    |   movel([0.490006, -1.325521, -2.603775, -0.783093, 1.570796, 2.060802],accel_mss,speed_ms,0,blend_radius_m)
    |   movel([0.490561, -1.327919, -2.602258, -0.782211, 1.570796, 2.061357],accel_mss,speed_ms,0,blend_radius_m)
    |   movel([0.493292, -1.324819, -2.604218, -0.783352, 1.570796, 2.064088],accel_mss,speed_ms,0,blend_radius_m)
    |   movel([0.496193, -1.321984, -2.605999, -0.784406, 1.570796, 2.066989],accel_mss,speed_ms,0,blend_radius_m)
    |   movel([0.499235, -1.319428, -2.607595, -0.785366, 1.570796, 2.070031],accel_mss,speed_ms,0,blend_radius_m)
    |   movel([0.502386, -1.317162, -2.609003, -0.786224, 1.570796, 2.073182],accel_mss,speed_ms,0,blend_radius_m)
    |   movel([0.505611, -1.315198, -2.610217, -0.786973, 1.570796, 2.076407],accel_mss,speed_ms,0,blend_radius_m)
    |   movel([0.508883, -1.313549, -2.611234, -0.787606, 1.570796, 2.079679],accel_mss,speed_ms,0,blend_radius_m)
    |   movel([0.512165, -1.312228, -2.612045, -0.788116, 1.570796, 2.082962],accel_mss,speed_ms,0,blend_radius_m)
    |   movel([0.515427, -1.311244, -2.612648, -0.788497, 1.570796, 2.086224],accel_mss,speed_ms,0,blend_radius_m)
    |   movel([0.518637, -1.310607, -2.613038, -0.788745, 1.570796, 2.089433],accel_mss,speed_ms,0,blend_radius_m)
    |   movel([0.521755, -1.310327, -2.613208, -0.788853, 1.570796, 2.092552],accel_mss,speed_ms,0,blend_radius_m)
    |   movel([0.524757, -1.310411, -2.613157, -0.788821, 1.570796, 2.095554],accel_mss,speed_ms,0,blend_radius_m)
    |   movel([0.527609, -1.310865, -2.612880, -0.788644, 1.570796, 2.098405],accel_mss,speed_ms,0,blend_radius_m)
    |   movel([0.530273, -1.311699, -2.612369, -0.788321, 1.570796, 2.101069],accel_mss,speed_ms,0,blend_radius_m)
    |   movel([0.532724, -1.312918, -2.611621, -0.787850, 1.570796, 2.103520],accel_mss,speed_ms,0,blend_radius_m)
    |   movel([0.534931, -1.314523, -2.610634, -0.787232, 1.570796, 2.105727],accel_mss,speed_ms,0,blend_radius_m)
    |   movel([0.536862, -1.316516, -2.609403, -0.786470, 1.570796, 2.107659],accel_mss,speed_ms,0,blend_radius_m)
    |   movel([0.538179, -1.318406, -2.608230, -0.785752, 1.570796, 2.108975],accel_mss,speed_ms,0,blend_radius_m)
    |   movel([0.539188, -1.320426, -2.606973, -0.784990, 1.570796, 2.109985],accel_mss,speed_ms,0,blend_radius_m)
    |   movel([0.539900, -1.322560, -2.605637, -0.784191, 1.570796, 2.110697],accel_mss,speed_ms,0,blend_radius_m)
    |   movel([0.540333, -1.324790, -2.604236, -0.783363, 1.570796, 2.111129],accel_mss,speed_ms,0,blend_radius_m)
    |   movel([0.540418, -1.329463, -2.601277, -0.781648, 1.570796, 2.111215],accel_mss,speed_ms,0,blend_radius_m)
    |   movel([0.539552, -1.334306, -2.598181, -0.779902, 1.570796, 2.110349],accel_mss,speed_ms,0,blend_radius_m)
    |   movel([0.537852, -1.339189, -2.595026, -0.778174, 1.570796, 2.108648],accel_mss,speed_ms,0,blend_radius_m)
    |   movel([0.535425, -1.343980, -2.591899, -0.776510, 1.570796, 2.106221],accel_mss,speed_ms,0,blend_radius_m)
    |   movel([0.532371, -1.348563, -2.588878, -0.774947, 1.570796, 2.103168],accel_mss,speed_ms,0,blend_radius_m)
    |   movel([0.528798, -1.352820, -2.586047, -0.773522, 1.570796, 2.099595],accel_mss,speed_ms,0,blend_radius_m)
    |   movel([0.524795, -1.356639, -2.583485, -0.772265, 1.570796, 2.095591],accel_mss,speed_ms,0,blend_radius_m)
    |   movel([0.520453, -1.359910, -2.581275, -0.771204, 1.570796, 2.091250],accel_mss,speed_ms,0,blend_radius_m)
    |   movel([0.515861, -1.362529, -2.579494, -0.770365, 1.570796, 2.086657],accel_mss,speed_ms,0,blend_radius_m)
    |   movel([0.513494, -1.363560, -2.578791, -0.770038, 1.570796, 2.084290],accel_mss,speed_ms,0,blend_radius_m)
    |   movel([0.511095, -1.364389, -2.578224, -0.769776, 1.570796, 2.081891],accel_mss,speed_ms,0,blend_radius_m)
    |   movel([0.508673, -1.364997, -2.577808, -0.769584, 1.570796, 2.079469],accel_mss,speed_ms,0,blend_radius_m)
    |   movel([0.506236, -1.365377, -2.577547, -0.769464, 1.570796, 2.077032],accel_mss,speed_ms,0,blend_radius_m)
    |   movel([0.503793, -1.365512, -2.577455, -0.769422, 1.570796, 2.074590],accel_mss,speed_ms,0,blend_radius_m)
    |   movel([0.501355, -1.365389, -2.577539, -0.769461, 1.570796, 2.072151],accel_mss,speed_ms,0,blend_radius_m)
    |   movel([0.498931, -1.364990, -2.577813, -0.769586, 1.570796, 2.069727],accel_mss,speed_ms,0,blend_radius_m)
    |   movel([0.496529, -1.364305, -2.578282, -0.769802, 1.570796, 2.067325],accel_mss,speed_ms,0,blend_radius_m)
    |   movel([0.494155, -1.363317, -2.578957, -0.770115, 1.570796, 2.064951],accel_mss,speed_ms,0,blend_radius_m)
    |   movel([0.491822, -1.362010, -2.579848, -0.770531, 1.570796, 2.062619],accel_mss,speed_ms,0,blend_radius_m)
    |   movel([0.490227, -1.360613, -2.580798, -0.770978, 1.570796, 2.061023],accel_mss,speed_ms,0,blend_radius_m)
    |   movel([0.486318, -1.356256, -2.583743, -0.772390, 1.570796, 2.057115],accel_mss,speed_ms,0,blend_radius_m)
    |   movel([0.483901, -1.352883, -2.586004, -0.773501, 1.570796, 2.054697],accel_mss,speed_ms,0,blend_radius_m)
    |   movel([0.481393, -1.348660, -2.588814, -0.774915, 1.570796, 2.052189],accel_mss,speed_ms,0,blend_radius_m)
    |   movel([0.478957, -1.343540, -2.592188, -0.776662, 1.570796, 2.049753],accel_mss,speed_ms,0,blend_radius_m)
    |   movel([0.476768, -1.337466, -2.596143, -0.778780, 1.570796, 2.047564],accel_mss,speed_ms,0,blend_radius_m)
    |   movel([0.475658, -1.332933, -2.599062, -0.780394, 1.570796, 2.046454],accel_mss,speed_ms,0,blend_radius_m)
    |   movel([0.475114, -1.328563, -2.601850, -0.781976, 1.570796, 2.045910],accel_mss,speed_ms,0,blend_radius_m)
    |   movel([0.475073, -1.324370, -2.604501, -0.783518, 1.570796, 2.045869],accel_mss,speed_ms,0,blend_radius_m)
    |   movel([0.475474, -1.320373, -2.607006, -0.785010, 1.570796, 2.046270],accel_mss,speed_ms,0,blend_radius_m)
    |   movel([0.476255, -1.316582, -2.609362, -0.786445, 1.570796, 2.047051],accel_mss,speed_ms,0,blend_radius_m)
    |   movel([0.477343, -1.313021, -2.611558, -0.787810, 1.570796, 2.048139],accel_mss,speed_ms,0,blend_radius_m)
    |   movel([0.478674, -1.309707, -2.613587, -0.789095, 1.570796, 2.049470],accel_mss,speed_ms,0,blend_radius_m)
    |   movel([0.480175, -1.306660, -2.615440, -0.790289, 1.570796, 2.050971],accel_mss,speed_ms,0,blend_radius_m)
    |   movel([0.483403, -1.301447, -2.618581, -0.792361, 1.570796, 2.054199],accel_mss,speed_ms,0,blend_radius_m)
    |   movel([0.486444, -1.297538, -2.620914, -0.793937, 1.570796, 2.057241],accel_mss,speed_ms,0,blend_radius_m)
    |   movel([0.488705, -1.295089, -2.622365, -0.794935, 1.570796, 2.059502],accel_mss,speed_ms,0,blend_radius_m)
    |   movel([0.489590, -1.294242, -2.622865, -0.795281, 1.570796, 2.060387],accel_mss,speed_ms,0,blend_radius_m)
    |   movel([0.493944, -1.290499, -2.625065, -0.796825, 1.570796, 2.064741],accel_mss,speed_ms,0,blend_radius_m)
    |   movel([0.498273, -1.287334, -2.626911, -0.798144, 1.570796, 2.069069],accel_mss,speed_ms,0,blend_radius_m)
    |   movel([0.502541, -1.284718, -2.628427, -0.799244, 1.570796, 2.073337],accel_mss,speed_ms,0,blend_radius_m)
    |   movel([0.506719, -1.282608, -2.629643, -0.800137, 1.570796, 2.077516],accel_mss,speed_ms,0,blend_radius_m)
    |   movel([0.510774, -1.280967, -2.630586, -0.800836, 1.570796, 2.081570],accel_mss,speed_ms,0,blend_radius_m)
    |   movel([0.514673, -1.279752, -2.631281, -0.801356, 1.570796, 2.085470],accel_mss,speed_ms,0,blend_radius_m)
    |   movel([0.518397, -1.278914, -2.631760, -0.801715, 1.570796, 2.089193],accel_mss,speed_ms,0,blend_radius_m)
    |   movel([0.521908, -1.278413, -2.632046, -0.801930, 1.570796, 2.092705],accel_mss,speed_ms,0,blend_radius_m)
    |   movel([0.528205, -1.278218, -2.632156, -0.802014, 1.570796, 2.099001],accel_mss,speed_ms,0,blend_radius_m)
    |   movel([0.533373, -1.278773, -2.631841, -0.801776, 1.570796, 2.104170],accel_mss,speed_ms,0,blend_radius_m)
    |   movel([0.537237, -1.279670, -2.631328, -0.801391, 1.570796, 2.108033],accel_mss,speed_ms,0,blend_radius_m)
    |   movel([0.539631, -1.280510, -2.630848, -0.801031, 1.570796, 2.110427],accel_mss,speed_ms,0,blend_radius_m)
    |   movel([0.545351, -1.282444, -2.629738, -0.800207, 1.570796, 2.116147],accel_mss,speed_ms,0,blend_radius_m)
    |   movel([0.551208, -1.285055, -2.628232, -0.799102, 1.570796, 2.122004],accel_mss,speed_ms,0,blend_radius_m)
    |   movel([0.557042, -1.287887, -2.626589, -0.797913, 1.570796, 2.127839],accel_mss,speed_ms,0,blend_radius_m)
    |   movel([0.562712, -1.290482, -2.625075, -0.796832, 1.570796, 2.133508],accel_mss,speed_ms,0,blend_radius_m)
    |   movel([0.568089, -1.292385, -2.623959, -0.796045, 1.570796, 2.138885],accel_mss,speed_ms,0,blend_radius_m)
    |   movel([0.570630, -1.292931, -2.623638, -0.795820, 1.570796, 2.141426],accel_mss,speed_ms,0,blend_radius_m)
    |   movel([0.573054, -1.293131, -2.623520, -0.795738, 1.570796, 2.143850],accel_mss,speed_ms,0,blend_radius_m)
    |   movel([0.575351, -1.292924, -2.623642, -0.795823, 1.570796, 2.146147],accel_mss,speed_ms,0,blend_radius_m)
    |   movel([0.577504, -1.292250, -2.624039, -0.796101, 1.570796, 2.148300],accel_mss,speed_ms,0,blend_radius_m)
    |   movel([0.579504, -1.291047, -2.624744, -0.796598, 1.570796, 2.150301],accel_mss,speed_ms,0,blend_radius_m)
    |   movel([0.581338, -1.289257, -2.625791, -0.797341, 1.570796, 2.152134],accel_mss,speed_ms,0,blend_radius_m)
    |   movel([0.582452, -1.287733, -2.626679, -0.797977, 1.570796, 2.153249],accel_mss,speed_ms,0,blend_radius_m)
    |   movel([0.583281, -1.286224, -2.627555, -0.798610, 1.570796, 2.154077],accel_mss,speed_ms,0,blend_radius_m)
    |   movel([0.584194, -1.283247, -2.629276, -0.799866, 1.570796, 2.154991],accel_mss,speed_ms,0,blend_radius_m)
    |   movel([0.584298, -1.280332, -2.630949, -0.801107, 1.570796, 2.155094],accel_mss,speed_ms,0,blend_radius_m)
    |   movel([0.583810, -1.277482, -2.632576, -0.802331, 1.570796, 2.154606],accel_mss,speed_ms,0,blend_radius_m)
    |   movel([0.581965, -1.272012, -2.635669, -0.804708, 1.570796, 2.152761],accel_mss,speed_ms,0,blend_radius_m)
    |   movel([0.581068, -1.269398, -2.637134, -0.805858, 1.570796, 2.151864],accel_mss,speed_ms,0,blend_radius_m)
    |   movel([0.580496, -1.266865, -2.638545, -0.806979, 1.570796, 2.151293],accel_mss,speed_ms,0,blend_radius_m)
    |   movel([0.580460, -1.262675, -2.640863, -0.808852, 1.570796, 2.151256],accel_mss,speed_ms,0,blend_radius_m)
    |   movel([0.581118, -1.257317, -2.643795, -0.811277, 1.570796, 2.151914],accel_mss,speed_ms,0,blend_radius_m)
    |   movel([0.582306, -1.251758, -2.646801, -0.813831, 1.570796, 2.153102],accel_mss,speed_ms,0,blend_radius_m)
    |   movel([0.583843, -1.247006, -2.649341, -0.816042, 1.570796, 2.154640],accel_mss,speed_ms,0,blend_radius_m)
    |   movel([0.585406, -1.244036, -2.650914, -0.817438, 1.570796, 2.156203],accel_mss,speed_ms,0,blend_radius_m)
    |   movel([0.587619, -1.240418, -2.652818, -0.819153, 1.570796, 2.158415],accel_mss,speed_ms,0,blend_radius_m)
    |   movel([0.589696, -1.236967, -2.654618, -0.820803, 1.570796, 2.160493],accel_mss,speed_ms,0,blend_radius_m)
    |   movel([0.590831, -1.234525, -2.655885, -0.821979, 1.570796, 2.161628],accel_mss,speed_ms,0,blend_radius_m)
    |   movel([0.590982, -1.232123, -2.657123, -0.823143, 1.570796, 2.161779],accel_mss,speed_ms,0,blend_radius_m)
    |   movel([0.590662, -1.229442, -2.658497, -0.824449, 1.570796, 2.161458],accel_mss,speed_ms,0,blend_radius_m)
    |   movel([0.590352, -1.226433, -2.660030, -0.825926, 1.570796, 2.161148],accel_mss,speed_ms,0,blend_radius_m)
    |   movel([0.590532, -1.223054, -2.661739, -0.827596, 1.570796, 2.161328],accel_mss,speed_ms,0,blend_radius_m)
    |   movel([0.591130, -1.220931, -2.662806, -0.828652, 1.570796, 2.161926],accel_mss,speed_ms,0,blend_radius_m)
    |   speed_ms = 0.003
    |   movel([0.591130, -1.213790, -2.659255, -0.839344, 1.570796, 2.161926],accel_mss,speed_ms,0,blend_radius_m)
    |   speed_ms = 0.05
    |   movel([0.591130, -1.186616, -2.644793, -0.880980, 1.570796, 2.161926],accel_mss,speed_ms,0,blend_radius_m)
    |   #M_RunCode9
    |   movel([0.476665, -1.280558, -2.594852, -0.836979, 1.570796, 2.047461],accel_mss,speed_ms,0,blend_radius_m)
    |   #M_RunCode3
    |   movel([0.476665, -1.306620, -2.608077, -0.797692, 1.570796, 2.047461],accel_mss,speed_ms,0,blend_radius_m)
    |   speed_ms = 0.003
    |   movel([0.476665, -1.313420, -2.611313, -0.787656, 1.570796, 2.047461],accel_mss,speed_ms,0,blend_radius_m)
    |   speed_ms = 0.02
    |   movel([0.470649, -1.312090, -2.612129, -0.788169, 1.570796, 2.041445],accel_mss,speed_ms,0,blend_radius_m)
    |   movel([0.464562, -1.311541, -2.612466, -0.788382, 1.570796, 2.035358],accel_mss,speed_ms,0,blend_radius_m)
    |   movel([0.458473, -1.311678, -2.612382, -0.788329, 1.570796, 2.029269],accel_mss,speed_ms,0,blend_radius_m)
    |   movel([0.452461, -1.312404, -2.611937, -0.788048, 1.570796, 2.023258],accel_mss,speed_ms,0,blend_radius_m)
    |   movel([0.446593, -1.313618, -2.611191, -0.787580, 1.570796, 2.017390],accel_mss,speed_ms,0,blend_radius_m)
    |   movel([0.440937, -1.315226, -2.610200, -0.786963, 1.570796, 2.011733],accel_mss,speed_ms,0,blend_radius_m)
    |   movel([0.435558, -1.317124, -2.609026, -0.786238, 1.570796, 2.006355],accel_mss,speed_ms,0,blend_radius_m)
    |   movel([0.430517, -1.319217, -2.607726, -0.785446, 1.570796, 2.001314],accel_mss,speed_ms,0,blend_radius_m)
    |   movel([0.425875, -1.321405, -2.606361, -0.784623, 1.570796, 1.996671],accel_mss,speed_ms,0,blend_radius_m)
    |   movel([0.421681, -1.323599, -2.604985, -0.783804, 1.570796, 1.992477],accel_mss,speed_ms,0,blend_radius_m)
    |   movel([0.414869, -1.327618, -2.602449, -0.782322, 1.570796, 1.985665],accel_mss,speed_ms,0,blend_radius_m)
    |   movel([0.410490, -1.330547, -2.600587, -0.781255, 1.570796, 1.981286],accel_mss,speed_ms,0,blend_radius_m)
    |   movel([0.408940, -1.331678, -2.599865, -0.780846, 1.570796, 1.979736],accel_mss,speed_ms,0,blend_radius_m)
    |   movel([0.406435, -1.333398, -2.598764, -0.780227, 1.570796, 1.977231],accel_mss,speed_ms,0,blend_radius_m)
    |   movel([0.400082, -1.338331, -2.595582, -0.778475, 1.570796, 1.970878],accel_mss,speed_ms,0,blend_radius_m)
    |   movel([0.396014, -1.341882, -2.593272, -0.777235, 1.570796, 1.966810],accel_mss,speed_ms,0,blend_radius_m)
    |   movel([0.391649, -1.346090, -2.590512, -0.775787, 1.570796, 1.962445],accel_mss,speed_ms,0,blend_radius_m)
    |   movel([0.387205, -1.350897, -2.587329, -0.774163, 1.570796, 1.958001],accel_mss,speed_ms,0,blend_radius_m)
    |   movel([0.382897, -1.356249, -2.583747, -0.772392, 1.570796, 1.953693],accel_mss,speed_ms,0,blend_radius_m)
    |   movel([0.378940, -1.362087, -2.579796, -0.770506, 1.570796, 1.949736],accel_mss,speed_ms,0,blend_radius_m)
    |   movel([0.375536, -1.368352, -2.575501, -0.768535, 1.570796, 1.946332],accel_mss,speed_ms,0,blend_radius_m)
    |   movel([0.374104, -1.371628, -2.573234, -0.767527, 1.570796, 1.944900],accel_mss,speed_ms,0,blend_radius_m)
    |   movel([0.372885, -1.374989, -2.570892, -0.766508, 1.570796, 1.943682],accel_mss,speed_ms,0,blend_radius_m)
    |   movel([0.371898, -1.378433, -2.568475, -0.765481, 1.570796, 1.942695],accel_mss,speed_ms,0,blend_radius_m)
    |   movel([0.371171, -1.381949, -2.565991, -0.764449, 1.570796, 1.941968],accel_mss,speed_ms,0,blend_radius_m)
    |   movel([0.370725, -1.385536, -2.563438, -0.763416, 1.570796, 1.941522],accel_mss,speed_ms,0,blend_radius_m)
    |   movel([0.370579, -1.389183, -2.560823, -0.762383, 1.570796, 1.941375],accel_mss,speed_ms,0,blend_radius_m)
    |   movel([0.370755, -1.392891, -2.558144, -0.761354, 1.570796, 1.941551],accel_mss,speed_ms,0,blend_radius_m)
    |   movel([0.371275, -1.396654, -2.555406, -0.760329, 1.570796, 1.942071],accel_mss,speed_ms,0,blend_radius_m)
    |   movel([0.372155, -1.400470, -2.552608, -0.759311, 1.570796, 1.942952],accel_mss,speed_ms,0,blend_radius_m)
    |   movel([0.373415, -1.404335, -2.549753, -0.758301, 1.570796, 1.944212],accel_mss,speed_ms,0,blend_radius_m)
    |   movel([0.375074, -1.408244, -2.546843, -0.757303, 1.570796, 1.945870],accel_mss,speed_ms,0,blend_radius_m)
    |   movel([0.377150, -1.412202, -2.543872, -0.756314, 1.570796, 1.947946],accel_mss,speed_ms,0,blend_radius_m)
    |   movel([0.377336, -1.412494, -2.543653, -0.756242, 1.570796, 1.948133],accel_mss,speed_ms,0,blend_radius_m)
    |   movel([0.380023, -1.415995, -2.541005, -0.755389, 1.570796, 1.950819],accel_mss,speed_ms,0,blend_radius_m)
    |   movel([0.382798, -1.419057, -2.538674, -0.754658, 1.570796, 1.953595],accel_mss,speed_ms,0,blend_radius_m)
    |   movel([0.385653, -1.421704, -2.536648, -0.754037, 1.570796, 1.956449],accel_mss,speed_ms,0,blend_radius_m)
    |   movel([0.388573, -1.423964, -2.534910, -0.753515, 1.570796, 1.959369],accel_mss,speed_ms,0,blend_radius_m)
    |   movel([0.391553, -1.425859, -2.533447, -0.753083, 1.570796, 1.962350],accel_mss,speed_ms,0,blend_radius_m)
    |   movel([0.394582, -1.427414, -2.532242, -0.752733, 1.570796, 1.965378],accel_mss,speed_ms,0,blend_radius_m)
    |   movel([0.397649, -1.428652, -2.531281, -0.752456, 1.570796, 1.968446],accel_mss,speed_ms,0,blend_radius_m)
    |   movel([0.400745, -1.429592, -2.530549, -0.752248, 1.570796, 1.971541],accel_mss,speed_ms,0,blend_radius_m)
    |   movel([0.403861, -1.430257, -2.530030, -0.752101, 1.570796, 1.974657],accel_mss,speed_ms,0,blend_radius_m)
    |   movel([0.406983, -1.430669, -2.529709, -0.752011, 1.570796, 1.977780],accel_mss,speed_ms,0,blend_radius_m)
    |   movel([0.410106, -1.430846, -2.529570, -0.751972, 1.570796, 1.980902],accel_mss,speed_ms,0,blend_radius_m)
    |   movel([0.413214, -1.430810, -2.529598, -0.751980, 1.570796, 1.984011],accel_mss,speed_ms,0,blend_radius_m)
    |   movel([0.419348, -1.430180, -2.530091, -0.752118, 1.570796, 1.990145],accel_mss,speed_ms,0,blend_radius_m)
    |   movel([0.425295, -1.428930, -2.531064, -0.752394, 1.570796, 1.996092],accel_mss,speed_ms,0,blend_radius_m)
    |   movel([0.430960, -1.427223, -2.532390, -0.752775, 1.570796, 2.001756],accel_mss,speed_ms,0,blend_radius_m)
    |   movel([0.436239, -1.425214, -2.533946, -0.753229, 1.570796, 2.007035],accel_mss,speed_ms,0,blend_radius_m)
    |   movel([0.441026, -1.423063, -2.535604, -0.753722, 1.570796, 2.011822],accel_mss,speed_ms,0,blend_radius_m)
    |   movel([0.445211, -1.420929, -2.537243, -0.754217, 1.570796, 2.016007],accel_mss,speed_ms,0,blend_radius_m)
    |   movel([0.451296, -1.417374, -2.539957, -0.755058, 1.570796, 2.022092],accel_mss,speed_ms,0,blend_radius_m)
    |   movel([0.453539, -1.415886, -2.541087, -0.755415, 1.570796, 2.024335],accel_mss,speed_ms,0,blend_radius_m)
    |   movel([0.454914, -1.415023, -2.541742, -0.755624, 1.570796, 2.025710],accel_mss,speed_ms,0,blend_radius_m)
    |   movel([0.458633, -1.412486, -2.543658, -0.756244, 1.570796, 2.029430],accel_mss,speed_ms,0,blend_radius_m)
    |   movel([0.464103, -1.408343, -2.546768, -0.757278, 1.570796, 2.034900],accel_mss,speed_ms,0,blend_radius_m)
    |   movel([0.470740, -1.402647, -2.551003, -0.758740, 1.570796, 2.041536],accel_mss,speed_ms,0,blend_radius_m)
    |   movel([0.474312, -1.399227, -2.553522, -0.759640, 1.570796, 2.045108],accel_mss,speed_ms,0,blend_radius_m)
    |   movel([0.477954, -1.395435, -2.556295, -0.760659, 1.570796, 2.048750],accel_mss,speed_ms,0,blend_radius_m)
    |   movel([0.481594, -1.391266, -2.559321, -0.761802, 1.570796, 2.052390],accel_mss,speed_ms,0,blend_radius_m)
    |   movel([0.485155, -1.386723, -2.562589, -0.763078, 1.570796, 2.055951],accel_mss,speed_ms,0,blend_radius_m)
    |   movel([0.488560, -1.381808, -2.566091, -0.764491, 1.570796, 2.059356],accel_mss,speed_ms,0,blend_radius_m)
    |   movel([0.491732, -1.376516, -2.569822, -0.766051, 1.570796, 2.062528],accel_mss,speed_ms,0,blend_radius_m)
    |   movel([0.494590, -1.370849, -2.573774, -0.767765, 1.570796, 2.065387],accel_mss,speed_ms,0,blend_radius_m)
    |   movel([0.497047, -1.364802, -2.577941, -0.769645, 1.570796, 2.067843],accel_mss,speed_ms,0,blend_radius_m)
    |   speed_ms = 0.003
    |   movel([0.497047, -1.358244, -2.574877, -0.779268, 1.570796, 2.067843],accel_mss,speed_ms,0,blend_radius_m)
    |   speed_ms = 0.05
    |   movel([0.497047, -1.333023, -2.562333, -0.817033, 1.570796, 2.067843],accel_mss,speed_ms,0,blend_radius_m)
    |   #M_RunCode9
    |   movel([0.471807, -1.327561, -2.565883, -0.818945, 1.570796, 2.042603],accel_mss,speed_ms,0,blend_radius_m)
    |   #M_RunCode3
    |   # logo 1
    |   movel([0.471807, -1.352876, -2.578497, -0.781015, 1.570796, 2.042603],accel_mss,speed_ms,0,blend_radius_m)
    |   speed_ms = 0.003
    |   movel([0.471807, -1.359461, -2.581579, -0.771349, 1.570796, 2.042603],accel_mss,speed_ms,0,blend_radius_m)
    |   speed_ms = 0.007
    |   movel([0.469753, -1.361986, -2.579865, -0.770539, 1.570796, 2.040549],accel_mss,speed_ms,0,blend_radius_m)
    |   movel([0.467378, -1.364236, -2.578329, -0.769824, 1.570796, 2.038174],accel_mss,speed_ms,0,blend_radius_m)
    |   movel([0.464761, -1.366165, -2.577007, -0.769217, 1.570796, 2.035557],accel_mss,speed_ms,0,blend_radius_m)
    |   movel([0.461981, -1.367726, -2.575933, -0.768730, 1.570796, 2.032778],accel_mss,speed_ms,0,blend_radius_m)
    |   movel([0.459114, -1.368870, -2.575144, -0.768375, 1.570796, 2.029910],accel_mss,speed_ms,0,blend_radius_m)
    |   movel([0.456235, -1.369551, -2.574673, -0.768165, 1.570796, 2.027032],accel_mss,speed_ms,0,blend_radius_m)
    |   movel([0.453420, -1.369720, -2.574557, -0.768113, 1.570796, 2.024216],accel_mss,speed_ms,0,blend_radius_m)
    |   movel([0.453380, -1.369716, -2.574559, -0.768114, 1.570796, 2.024176],accel_mss,speed_ms,0,blend_radius_m)
    |   movel([0.447352, -1.369503, -2.574707, -0.768180, 1.570796, 2.018149],accel_mss,speed_ms,0,blend_radius_m)
    |   movel([0.443007, -1.378673, -2.568306, -0.765410, 1.570796, 2.013804],accel_mss,speed_ms,0,blend_radius_m)
    |   movel([0.435809, -1.378470, -2.568449, -0.765470, 1.570796, 2.006605],accel_mss,speed_ms,0,blend_radius_m)
    |   movel([0.448034, -1.352401, -2.586327, -0.773661, 1.570796, 2.018830],accel_mss,speed_ms,0,blend_radius_m)
    |   movel([0.455424, -1.352614, -2.586184, -0.773591, 1.570796, 2.026221],accel_mss,speed_ms,0,blend_radius_m)
    |   movel([0.450911, -1.362037, -2.579830, -0.770522, 1.570796, 2.021708],accel_mss,speed_ms,0,blend_radius_m)
    |   movel([0.457056, -1.362252, -2.579683, -0.770454, 1.570796, 2.027852],accel_mss,speed_ms,0,blend_radius_m)
    |   movel([0.458332, -1.362171, -2.579738, -0.770479, 1.570796, 2.029128],accel_mss,speed_ms,0,blend_radius_m)
    |   movel([0.459648, -1.361851, -2.579957, -0.770582, 1.570796, 2.030444],accel_mss,speed_ms,0,blend_radius_m)
    |   movel([0.460964, -1.361314, -2.580321, -0.770753, 1.570796, 2.031760],accel_mss,speed_ms,0,blend_radius_m)
    |   movel([0.462242, -1.360591, -2.580813, -0.770985, 1.570796, 2.033038],accel_mss,speed_ms,0,blend_radius_m)
    |   movel([0.463445, -1.359699, -2.581418, -0.771272, 1.570796, 2.034241],accel_mss,speed_ms,0,blend_radius_m)
    |   movel([0.464532, -1.358666, -2.582117, -0.771606, 1.570796, 2.035329],accel_mss,speed_ms,0,blend_radius_m)
    |   movel([0.465466, -1.357515, -2.582895, -0.771979, 1.570796, 2.036262],accel_mss,speed_ms,0,blend_radius_m)
    |   movel([0.466207, -1.356275, -2.583730, -0.772384, 1.570796, 2.037003],accel_mss,speed_ms,0,blend_radius_m)
    |   movel([0.466698, -1.355017, -2.584575, -0.772796, 1.570796, 2.037494],accel_mss,speed_ms,0,blend_radius_m)
    |   movel([0.466925, -1.353822, -2.585377, -0.773190, 1.570796, 2.037721],accel_mss,speed_ms,0,blend_radius_m)
    |   movel([0.466616, -1.351745, -2.586764, -0.773880, 1.570796, 2.037412],accel_mss,speed_ms,0,blend_radius_m)
    |   movel([0.466103, -1.350922, -2.587312, -0.774155, 1.570796, 2.036899],accel_mss,speed_ms,0,blend_radius_m)
    |   movel([0.465361, -1.350281, -2.587739, -0.774369, 1.570796, 2.036158],accel_mss,speed_ms,0,blend_radius_m)
    |   movel([0.464402, -1.349855, -2.588022, -0.774512, 1.570796, 2.035199],accel_mss,speed_ms,0,blend_radius_m)
    |   movel([0.463240, -1.349675, -2.588141, -0.774573, 1.570796, 2.034037],accel_mss,speed_ms,0,blend_radius_m)
    |   movel([0.438898, -1.349022, -2.588575, -0.774793, 1.570796, 2.009694],accel_mss,speed_ms,0,blend_radius_m)
    |   movel([0.438801, -1.346776, -2.590060, -0.775553, 1.570796, 2.009597],accel_mss,speed_ms,0,blend_radius_m)
    |   movel([0.438301, -1.344731, -2.591406, -0.776252, 1.570796, 2.009097],accel_mss,speed_ms,0,blend_radius_m)
    |   movel([0.437406, -1.342923, -2.592592, -0.776875, 1.570796, 2.008203],accel_mss,speed_ms,0,blend_radius_m)
    |   movel([0.436133, -1.341382, -2.593598, -0.777408, 1.570796, 2.006929],accel_mss,speed_ms,0,blend_radius_m)
    |   movel([0.466821, -1.342114, -2.593121, -0.777154, 1.570796, 2.037618],accel_mss,speed_ms,0,blend_radius_m)
    |   movel([0.469435, -1.342515, -2.592859, -0.777016, 1.570796, 2.040231],accel_mss,speed_ms,0,blend_radius_m)
    |   movel([0.471592, -1.343449, -2.592247, -0.776693, 1.570796, 2.042388],accel_mss,speed_ms,0,blend_radius_m)
    |   movel([0.473260, -1.344857, -2.591323, -0.776209, 1.570796, 2.044056],accel_mss,speed_ms,0,blend_radius_m)
    |   movel([0.474412, -1.346673, -2.590127, -0.775588, 1.570796, 2.045208],accel_mss,speed_ms,0,blend_radius_m)
    |   movel([0.475032, -1.348830, -2.588701, -0.774857, 1.570796, 2.045829],accel_mss,speed_ms,0,blend_radius_m)
    |   movel([0.475093, -1.351262, -2.587086, -0.774041, 1.570796, 2.045889],accel_mss,speed_ms,0,blend_radius_m)
    |   movel([0.474576, -1.353911, -2.585317, -0.773161, 1.570796, 2.045372],accel_mss,speed_ms,0,blend_radius_m)
    |   movel([0.473459, -1.356706, -2.583440, -0.772243, 1.570796, 2.044255],accel_mss,speed_ms,0,blend_radius_m)
    |   movel([0.471807, -1.359461, -2.581579, -0.771349, 1.570796, 2.042603],accel_mss,speed_ms,0,blend_radius_m)
    |   speed_ms = 0.003
    |   movel([0.471807, -1.352876, -2.578497, -0.781015, 1.570796, 2.042603],accel_mss,speed_ms,0,blend_radius_m)
    |   speed_ms = 0.05
    |   movel([0.471807, -1.327561, -2.565883, -0.818945, 1.570796, 2.042603],accel_mss,speed_ms,0,blend_radius_m)
    |   #M_RunCode9
    |   movel([0.468567, -1.334790, -2.561176, -0.816423, 1.570796, 2.039363],accel_mss,speed_ms,0,blend_radius_m)
    |   #M_RunCode3
    |   # logo 2
    |   movel([0.468567, -1.359981, -2.573697, -0.778711, 1.570796, 2.039363],accel_mss,speed_ms,0,blend_radius_m)
    |   speed_ms = 0.003
    |   movel([0.468567, -1.366530, -2.576756, -0.769103, 1.570796, 2.039363],accel_mss,speed_ms,0,blend_radius_m)
    |   speed_ms = 0.007
    |   movel([0.454098, -1.395970, -2.555905, -0.760513, 1.570796, 2.024894],accel_mss,speed_ms,0,blend_radius_m)
    |   movel([0.452569, -1.398555, -2.554015, -0.759819, 1.570796, 2.023365],accel_mss,speed_ms,0,blend_radius_m)
    |   movel([0.450645, -1.400927, -2.552272, -0.759190, 1.570796, 2.021441],accel_mss,speed_ms,0,blend_radius_m)
    |   movel([0.448403, -1.403043, -2.550710, -0.758636, 1.570796, 2.019200],accel_mss,speed_ms,0,blend_radius_m)
    |   movel([0.445920, -1.404860, -2.549363, -0.758166, 1.570796, 2.016717],accel_mss,speed_ms,0,blend_radius_m)
    |   movel([0.443273, -1.406329, -2.548271, -0.757789, 1.570796, 2.014070],accel_mss,speed_ms,0,blend_radius_m)
    |   movel([0.440533, -1.407407, -2.547468, -0.757515, 1.570796, 2.011329],accel_mss,speed_ms,0,blend_radius_m)
    |   movel([0.437776, -1.408050, -2.546988, -0.757352, 1.570796, 2.008573],accel_mss,speed_ms,0,blend_radius_m)
    |   movel([0.435071, -1.408210, -2.546868, -0.757311, 1.570796, 2.005868],accel_mss,speed_ms,0,blend_radius_m)
    |   movel([0.432602, -1.407864, -2.547126, -0.757399, 1.570796, 2.003398],accel_mss,speed_ms,0,blend_radius_m)
    |   movel([0.430530, -1.407048, -2.547735, -0.757606, 1.570796, 2.001327],accel_mss,speed_ms,0,blend_radius_m)
    |   movel([0.428882, -1.405812, -2.548656, -0.757921, 1.570796, 1.999679],accel_mss,speed_ms,0,blend_radius_m)
    |   movel([0.427691, -1.404201, -2.549852, -0.758336, 1.570796, 1.998487],accel_mss,speed_ms,0,blend_radius_m)
    |   movel([0.426984, -1.402267, -2.551283, -0.758839, 1.570796, 1.997780],accel_mss,speed_ms,0,blend_radius_m)
    |   movel([0.426790, -1.400058, -2.552912, -0.759420, 1.570796, 1.997586],accel_mss,speed_ms,0,blend_radius_m)
    |   movel([0.427145, -1.397620, -2.554700, -0.760069, 1.570796, 1.997942],accel_mss,speed_ms,0,blend_radius_m)
    |   movel([0.428083, -1.395004, -2.556609, -0.760776, 1.570796, 1.998879],accel_mss,speed_ms,0,blend_radius_m)
    |   movel([0.428098, -1.394971, -2.556634, -0.760785, 1.570796, 1.998895],accel_mss,speed_ms,0,blend_radius_m)
    |   movel([0.430810, -1.389093, -2.560887, -0.762408, 1.570796, 2.001607],accel_mss,speed_ms,0,blend_radius_m)
    |   movel([0.421778, -1.388923, -2.561010, -0.762456, 1.570796, 1.992574],accel_mss,speed_ms,0,blend_radius_m)
    |   movel([0.425026, -1.381773, -2.566115, -0.764501, 1.570796, 1.995823],accel_mss,speed_ms,0,blend_radius_m)
    |   movel([0.450416, -1.382475, -2.565618, -0.764297, 1.570796, 2.021212],accel_mss,speed_ms,0,blend_radius_m)
    |   movel([0.446998, -1.389600, -2.560522, -0.762266, 1.570796, 2.017795],accel_mss,speed_ms,0,blend_radius_m)
    |   movel([0.438038, -1.389283, -2.560751, -0.762355, 1.570796, 2.008834],accel_mss,speed_ms,0,blend_radius_m)
    |   movel([0.435252, -1.395226, -2.556448, -0.760715, 1.570796, 2.006048],accel_mss,speed_ms,0,blend_radius_m)
    |   movel([0.434826, -1.396403, -2.555590, -0.760397, 1.570796, 2.005622],accel_mss,speed_ms,0,blend_radius_m)
    |   movel([0.434659, -1.397511, -2.554779, -0.760098, 1.570796, 2.005456],accel_mss,speed_ms,0,blend_radius_m)
    |   movel([0.434744, -1.398526, -2.554037, -0.759827, 1.570796, 2.005540],accel_mss,speed_ms,0,blend_radius_m)
    |   movel([0.435062, -1.399421, -2.553380, -0.759589, 1.570796, 2.005858],accel_mss,speed_ms,0,blend_radius_m)
    |   movel([0.435600, -1.400169, -2.552830, -0.759390, 1.570796, 2.006396],accel_mss,speed_ms,0,blend_radius_m)
    |   movel([0.436345, -1.400747, -2.552404, -0.759238, 1.570796, 2.007142],accel_mss,speed_ms,0,blend_radius_m)
    |   movel([0.437284, -1.401127, -2.552124, -0.759138, 1.570796, 2.008080],accel_mss,speed_ms,0,blend_radius_m)
    |   movel([0.438399, -1.401288, -2.552006, -0.759095, 1.570796, 2.009196],accel_mss,speed_ms,0,blend_radius_m)
    |   movel([0.439626, -1.401217, -2.552058, -0.759114, 1.570796, 2.010423],accel_mss,speed_ms,0,blend_radius_m)
    |   movel([0.440882, -1.400925, -2.552273, -0.759191, 1.570796, 2.011679],accel_mss,speed_ms,0,blend_radius_m)
    |   movel([0.443349, -1.399765, -2.553127, -0.759497, 1.570796, 2.014145],accel_mss,speed_ms,0,blend_radius_m)
    |   movel([0.444486, -1.398941, -2.553732, -0.759716, 1.570796, 2.015282],accel_mss,speed_ms,0,blend_radius_m)
    |   movel([0.445509, -1.397981, -2.554435, -0.759972, 1.570796, 2.016305],accel_mss,speed_ms,0,blend_radius_m)
    |   movel([0.446378, -1.396910, -2.555219, -0.760260, 1.570796, 2.017175],accel_mss,speed_ms,0,blend_radius_m)
    |   movel([0.447063, -1.395746, -2.556069, -0.760574, 1.570796, 2.017860],accel_mss,speed_ms,0,blend_radius_m)
    |   movel([0.458426, -1.372274, -2.572785, -0.767330, 1.570796, 2.029222],accel_mss,speed_ms,0,blend_radius_m)
    |   movel([0.461074, -1.371271, -2.573481, -0.767636, 1.570796, 2.031870],accel_mss,speed_ms,0,blend_radius_m)
    |   movel([0.463676, -1.369963, -2.574388, -0.768038, 1.570796, 2.034473],accel_mss,speed_ms,0,blend_radius_m)
    |   movel([0.466188, -1.368374, -2.575486, -0.768529, 1.570796, 2.036984],accel_mss,speed_ms,0,blend_radius_m)
    |   movel([0.468567, -1.366530, -2.576756, -0.769103, 1.570796, 2.039363],accel_mss,speed_ms,0,blend_radius_m)
    |   speed_ms = 0.003
    |   movel([0.468567, -1.359981, -2.573697, -0.778711, 1.570796, 2.039363],accel_mss,speed_ms,0,blend_radius_m)
    |   speed_ms = 0.05
    |   movel([0.468567, -1.334790, -2.561176, -0.816423, 1.570796, 2.039363],accel_mss,speed_ms,0,blend_radius_m)
    |   #M_RunCode9
    |   movel([0.425741, -1.340932, -2.557122, -0.814335, 1.570796, 1.996537],accel_mss,speed_ms,0,blend_radius_m)
    |   #M_RunCode3
    |   # logo 3
    |   movel([0.425741, -1.366016, -2.569564, -0.776808, 1.570796, 1.996537],accel_mss,speed_ms,0,blend_radius_m)
    |   speed_ms = 0.003
    |   movel([0.425741, -1.372535, -2.572603, -0.767250, 1.570796, 1.996537],accel_mss,speed_ms,0,blend_radius_m)
    |   speed_ms = 0.007
    |   movel([0.414358, -1.397807, -2.554563, -0.760019, 1.570796, 1.985154],accel_mss,speed_ms,0,blend_radius_m)
    |   movel([0.407219, -1.397755, -2.554601, -0.760033, 1.570796, 1.978015],accel_mss,speed_ms,0,blend_radius_m)
    |   movel([0.411153, -1.388853, -2.561060, -0.762476, 1.570796, 1.981950],accel_mss,speed_ms,0,blend_radius_m)
    |   movel([0.405078, -1.388847, -2.561065, -0.762478, 1.570796, 1.975874],accel_mss,speed_ms,0,blend_radius_m)
    |   movel([0.403816, -1.388971, -2.560975, -0.762443, 1.570796, 1.974613],accel_mss,speed_ms,0,blend_radius_m)
    |   movel([0.402531, -1.389327, -2.560719, -0.762343, 1.570796, 1.973328],accel_mss,speed_ms,0,blend_radius_m)
    |   movel([0.401264, -1.389886, -2.560316, -0.762186, 1.570796, 1.972060],accel_mss,speed_ms,0,blend_radius_m)
    |   movel([0.400049, -1.390622, -2.559786, -0.761981, 1.570796, 1.970845],accel_mss,speed_ms,0,blend_radius_m)
    |   movel([0.398925, -1.391508, -2.559145, -0.761735, 1.570796, 1.969721],accel_mss,speed_ms,0,blend_radius_m)
    |   movel([0.397929, -1.392517, -2.558415, -0.761456, 1.570796, 1.968725],accel_mss,speed_ms,0,blend_radius_m)
    |   movel([0.397098, -1.393625, -2.557612, -0.761152, 1.570796, 1.967894],accel_mss,speed_ms,0,blend_radius_m)
    |   movel([0.396471, -1.394803, -2.556756, -0.760830, 1.570796, 1.967267],accel_mss,speed_ms,0,blend_radius_m)
    |   movel([0.396087, -1.395979, -2.555899, -0.760511, 1.570796, 1.966884],accel_mss,speed_ms,0,blend_radius_m)
    |   movel([0.395960, -1.397078, -2.555097, -0.760215, 1.570796, 1.966756],accel_mss,speed_ms,0,blend_radius_m)
    |   movel([0.396427, -1.398949, -2.553726, -0.759714, 1.570796, 1.967224],accel_mss,speed_ms,0,blend_radius_m)
    |   movel([0.396993, -1.399671, -2.553196, -0.759522, 1.570796, 1.967789],accel_mss,speed_ms,0,blend_radius_m)
    |   movel([0.397761, -1.400218, -2.552794, -0.759377, 1.570796, 1.968557],accel_mss,speed_ms,0,blend_radius_m)
    |   movel([0.398717, -1.400565, -2.552538, -0.759286, 1.570796, 1.969514],accel_mss,speed_ms,0,blend_radius_m)
    |   movel([0.399855, -1.400685, -2.552450, -0.759254, 1.570796, 1.970651],accel_mss,speed_ms,0,blend_radius_m)
    |   movel([0.423157, -1.400895, -2.552295, -0.759199, 1.570796, 1.993953],accel_mss,speed_ms,0,blend_radius_m)
    |   movel([0.423288, -1.402968, -2.550765, -0.758656, 1.570796, 1.994084],accel_mss,speed_ms,0,blend_radius_m)
    |   movel([0.423793, -1.404846, -2.549373, -0.758169, 1.570796, 1.994590],accel_mss,speed_ms,0,blend_radius_m)
    |   movel([0.424654, -1.406506, -2.548139, -0.757744, 1.570796, 1.995450],accel_mss,speed_ms,0,blend_radius_m)
    |   movel([0.425854, -1.407923, -2.547082, -0.757384, 1.570796, 1.996650],accel_mss,speed_ms,0,blend_radius_m)
    |   movel([0.396983, -1.407574, -2.547342, -0.757472, 1.570796, 1.967780],accel_mss,speed_ms,0,blend_radius_m)
    |   movel([0.394459, -1.407325, -2.547529, -0.757535, 1.570796, 1.965255],accel_mss,speed_ms,0,blend_radius_m)
    |   movel([0.392320, -1.406597, -2.548071, -0.757721, 1.570796, 1.963116],accel_mss,speed_ms,0,blend_radius_m)
    |   movel([0.390594, -1.405436, -2.548935, -0.758018, 1.570796, 1.961390],accel_mss,speed_ms,0,blend_radius_m)
    |   movel([0.389313, -1.403892, -2.550081, -0.758416, 1.570796, 1.960109],accel_mss,speed_ms,0,blend_radius_m)
    |   movel([0.388507, -1.402011, -2.551473, -0.758906, 1.570796, 1.959304],accel_mss,speed_ms,0,blend_radius_m)
    |   movel([0.388210, -1.399839, -2.553072, -0.759478, 1.570796, 1.959007],accel_mss,speed_ms,0,blend_radius_m)
    |   movel([0.388459, -1.397427, -2.554841, -0.760121, 1.570796, 1.959255],accel_mss,speed_ms,0,blend_radius_m)
    |   movel([0.389288, -1.394822, -2.556742, -0.760825, 1.570796, 1.960085],accel_mss,speed_ms,0,blend_radius_m)
    |   movel([0.390663, -1.392200, -2.558645, -0.761544, 1.570796, 1.961459],accel_mss,speed_ms,0,blend_radius_m)
    |   movel([0.392475, -1.389739, -2.560422, -0.762228, 1.570796, 1.963271],accel_mss,speed_ms,0,blend_radius_m)
    |   movel([0.394652, -1.387498, -2.562033, -0.762858, 1.570796, 1.965448],accel_mss,speed_ms,0,blend_radius_m)
    |   movel([0.397120, -1.385535, -2.563438, -0.763416, 1.570796, 1.967916],accel_mss,speed_ms,0,blend_radius_m)
    |   movel([0.399796, -1.383903, -2.564602, -0.763884, 1.570796, 1.970592],accel_mss,speed_ms,0,blend_radius_m)
    |   movel([0.402603, -1.382666, -2.565482, -0.764241, 1.570796, 1.973399],accel_mss,speed_ms,0,blend_radius_m)
    |   movel([0.405459, -1.381879, -2.566040, -0.764470, 1.570796, 1.976255],accel_mss,speed_ms,0,blend_radius_m)
    |   movel([0.408280, -1.381600, -2.566238, -0.764551, 1.570796, 1.979076],accel_mss,speed_ms,0,blend_radius_m)
    |   movel([0.408310, -1.381609, -2.566231, -0.764548, 1.570796, 1.979107],accel_mss,speed_ms,0,blend_radius_m)
    |   movel([0.414363, -1.381607, -2.566233, -0.764549, 1.570796, 1.985159],accel_mss,speed_ms,0,blend_radius_m)
    |   movel([0.418427, -1.372480, -2.572642, -0.767267, 1.570796, 1.989224],accel_mss,speed_ms,0,blend_radius_m)
    |   movel([0.425741, -1.372535, -2.572603, -0.767250, 1.570796, 1.996537],accel_mss,speed_ms,0,blend_radius_m)
    |   speed_ms = 0.003
    |   movel([0.425741, -1.366016, -2.569564, -0.776808, 1.570796, 1.996537],accel_mss,speed_ms,0,blend_radius_m)
    |   speed_ms = 0.05
    |   movel([0.425741, -1.340932, -2.557122, -0.814335, 1.570796, 1.996537],accel_mss,speed_ms,0,blend_radius_m)
    |   #M_RunCode9
    |   movel([0.436628, -1.337490, -2.559400, -0.815499, 1.570796, 2.007425],accel_mss,speed_ms,0,blend_radius_m)
    |   #M_RunCode3
    |   # logo 4
    |   movel([0.436628, -1.362634, -2.571887, -0.777868, 1.570796, 2.007425],accel_mss,speed_ms,0,blend_radius_m)
    |   speed_ms = 0.003
    |   movel([0.436628, -1.369170, -2.574937, -0.768282, 1.570796, 2.007425],accel_mss,speed_ms,0,blend_radius_m)
    |   speed_ms = 0.007
    |   movel([0.410669, -1.368971, -2.575074, -0.768344, 1.570796, 1.981465],accel_mss,speed_ms,0,blend_radius_m)
    |   movel([0.413915, -1.361592, -2.580132, -0.770664, 1.570796, 1.984712],accel_mss,speed_ms,0,blend_radius_m)
    |   movel([0.423280, -1.361588, -2.580136, -0.770666, 1.570796, 1.994076],accel_mss,speed_ms,0,blend_radius_m)
    |   movel([0.426109, -1.355308, -2.584381, -0.772701, 1.570796, 1.996905],accel_mss,speed_ms,0,blend_radius_m)
    |   movel([0.426548, -1.354054, -2.585221, -0.773114, 1.570796, 1.997344],accel_mss,speed_ms,0,blend_radius_m)
    |   movel([0.426709, -1.352877, -2.586009, -0.773503, 1.570796, 1.997505],accel_mss,speed_ms,0,blend_radius_m)
    |   movel([0.426607, -1.351805, -2.586724, -0.773860, 1.570796, 1.997404],accel_mss,speed_ms,0,blend_radius_m)
    |   movel([0.426259, -1.350864, -2.587351, -0.774174, 1.570796, 1.997056],accel_mss,speed_ms,0,blend_radius_m)
    |   movel([0.425677, -1.350084, -2.587870, -0.774435, 1.570796, 1.996473],accel_mss,speed_ms,0,blend_radius_m)
    |   movel([0.424876, -1.349492, -2.588263, -0.774634, 1.570796, 1.995672],accel_mss,speed_ms,0,blend_radius_m)
    |   movel([0.423867, -1.349118, -2.588511, -0.774760, 1.570796, 1.994663],accel_mss,speed_ms,0,blend_radius_m)
    |   movel([0.422670, -1.348989, -2.588596, -0.774804, 1.570796, 1.993466],accel_mss,speed_ms,0,blend_radius_m)
    |   movel([0.421357, -1.349119, -2.588510, -0.774760, 1.570796, 1.992153],accel_mss,speed_ms,0,blend_radius_m)
    |   movel([0.420014, -1.349489, -2.588264, -0.774635, 1.570796, 1.990810],accel_mss,speed_ms,0,blend_radius_m)
    |   movel([0.417397, -1.350842, -2.587366, -0.774181, 1.570796, 1.988193],accel_mss,speed_ms,0,blend_radius_m)
    |   movel([0.416208, -1.351770, -2.586747, -0.773871, 1.570796, 1.987004],accel_mss,speed_ms,0,blend_radius_m)
    |   movel([0.415147, -1.352834, -2.586038, -0.773518, 1.570796, 1.985944],accel_mss,speed_ms,0,blend_radius_m)
    |   movel([0.414258, -1.354005, -2.585254, -0.773130, 1.570796, 1.985054],accel_mss,speed_ms,0,blend_radius_m)
    |   movel([0.413573, -1.355259, -2.584413, -0.772717, 1.570796, 1.984369],accel_mss,speed_ms,0,blend_radius_m)
    |   movel([0.403071, -1.379378, -2.567809, -0.765202, 1.570796, 1.973868],accel_mss,speed_ms,0,blend_radius_m)
    |   movel([0.400446, -1.380488, -2.567025, -0.764876, 1.570796, 1.971243],accel_mss,speed_ms,0,blend_radius_m)
    |   movel([0.397906, -1.381887, -2.566034, -0.764467, 1.570796, 1.968703],accel_mss,speed_ms,0,blend_radius_m)
    |   movel([0.395495, -1.383549, -2.564854, -0.763986, 1.570796, 1.966291],accel_mss,speed_ms,0,blend_radius_m)
    |   movel([0.393250, -1.385439, -2.563507, -0.763443, 1.570796, 1.964047],accel_mss,speed_ms,0,blend_radius_m)
    |   movel([0.406066, -1.355455, -2.584281, -0.772652, 1.570796, 1.976862],accel_mss,speed_ms,0,blend_radius_m)
    |   movel([0.407553, -1.352663, -2.586152, -0.773574, 1.570796, 1.978349],accel_mss,speed_ms,0,blend_radius_m)
    |   movel([0.409496, -1.350040, -2.587899, -0.774450, 1.570796, 1.980293],accel_mss,speed_ms,0,blend_radius_m)
    |   movel([0.411817, -1.347654, -2.589480, -0.775255, 1.570796, 1.982614],accel_mss,speed_ms,0,blend_radius_m)
    |   movel([0.414431, -1.345562, -2.590860, -0.775967, 1.570796, 1.985227],accel_mss,speed_ms,0,blend_radius_m)
    |   movel([0.417258, -1.343823, -2.592002, -0.776564, 1.570796, 1.988055],accel_mss,speed_ms,0,blend_radius_m)
    |   movel([0.420212, -1.342505, -2.592865, -0.777019, 1.570796, 1.991009],accel_mss,speed_ms,0,blend_radius_m)
    |   movel([0.423204, -1.341668, -2.593412, -0.777309, 1.570796, 1.994001],accel_mss,speed_ms,0,blend_radius_m)
    |   movel([0.426148, -1.341370, -2.593607, -0.777413, 1.570796, 1.996944],accel_mss,speed_ms,0,blend_radius_m)
    |   movel([0.428833, -1.341652, -2.593422, -0.777315, 1.570796, 1.999629],accel_mss,speed_ms,0,blend_radius_m)
    |   movel([0.431076, -1.342480, -2.592881, -0.777028, 1.570796, 2.001872],accel_mss,speed_ms,0,blend_radius_m)
    |   movel([0.432845, -1.343789, -2.592024, -0.776576, 1.570796, 2.003642],accel_mss,speed_ms,0,blend_radius_m)
    |   movel([0.434115, -1.345518, -2.590888, -0.775982, 1.570796, 2.004911],accel_mss,speed_ms,0,blend_radius_m)
    |   movel([0.434854, -1.347605, -2.589512, -0.775272, 1.570796, 2.005650],accel_mss,speed_ms,0,blend_radius_m)
    |   movel([0.435035, -1.349988, -2.587933, -0.774468, 1.570796, 2.005831],accel_mss,speed_ms,0,blend_radius_m)
    |   movel([0.434637, -1.352608, -2.586189, -0.773593, 1.570796, 2.005434],accel_mss,speed_ms,0,blend_radius_m)
    |   movel([0.433633, -1.355402, -2.584317, -0.772670, 1.570796, 2.004429],accel_mss,speed_ms,0,blend_radius_m)
    |   movel([0.433615, -1.355439, -2.584292, -0.772658, 1.570796, 2.004412],accel_mss,speed_ms,0,blend_radius_m)
    |   movel([0.430777, -1.361647, -2.580095, -0.770647, 1.570796, 2.001573],accel_mss,speed_ms,0,blend_radius_m)
    |   movel([0.440059, -1.361800, -2.579991, -0.770598, 1.570796, 2.010855],accel_mss,speed_ms,0,blend_radius_m)
    |   movel([0.436628, -1.369170, -2.574937, -0.768282, 1.570796, 2.007425],accel_mss,speed_ms,0,blend_radius_m)
    |   speed_ms = 0.003
    |   movel([0.436628, -1.362634, -2.571887, -0.777868, 1.570796, 2.007425],accel_mss,speed_ms,0,blend_radius_m)
    |   speed_ms = 0.05
    |   movel([0.436628, -1.337490, -2.559400, -0.815499, 1.570796, 2.007425],accel_mss,speed_ms,0,blend_radius_m)
    |   #M_RunCode9
    |   movel([0.384728, -1.390650, -2.522431, -0.799308, 1.570796, 1.955525],accel_mss,speed_ms,0,blend_radius_m)
    |   #M_RunCode3
    |   movel([0.384728, -1.414816, -2.534247, -0.763326, 1.570796, 1.955525],accel_mss,speed_ms,0,blend_radius_m)
    |   speed_ms = 0.003
    |   movel([0.384728, -1.421077, -2.537129, -0.754183, 1.570796, 1.955525],accel_mss,speed_ms,0,blend_radius_m)
    |   speed_ms = 0.02
    |   movel([0.387538, -1.423816, -2.535024, -0.753549, 1.570796, 1.958335],accel_mss,speed_ms,0,blend_radius_m)
    |   movel([0.391957, -1.427017, -2.532550, -0.752822, 1.570796, 1.962754],accel_mss,speed_ms,0,blend_radius_m)
    |   movel([0.397492, -1.430394, -2.529923, -0.752071, 1.570796, 1.968288],accel_mss,speed_ms,0,blend_radius_m)
    |   movel([0.403670, -1.433660, -2.527367, -0.751362, 1.570796, 1.974466],accel_mss,speed_ms,0,blend_radius_m)
    |   movel([0.410034, -1.436512, -2.525121, -0.750756, 1.570796, 1.980830],accel_mss,speed_ms,0,blend_radius_m)
    |   movel([0.416148, -1.438638, -2.523439, -0.750312, 1.570796, 1.986944],accel_mss,speed_ms,0,blend_radius_m)
    |   movel([0.418982, -1.439329, -2.522891, -0.750169, 1.570796, 1.989778],accel_mss,speed_ms,0,blend_radius_m)
    |   movel([0.421597, -1.439718, -2.522582, -0.750089, 1.570796, 1.992393],accel_mss,speed_ms,0,blend_radius_m)
    |   movel([0.423945, -1.439759, -2.522549, -0.750080, 1.570796, 1.994742],accel_mss,speed_ms,0,blend_radius_m)
    |   movel([0.425973, -1.439412, -2.522825, -0.750152, 1.570796, 1.996770],accel_mss,speed_ms,0,blend_radius_m)
    |   movel([0.427534, -1.438680, -2.523406, -0.750303, 1.570796, 1.998330],accel_mss,speed_ms,0,blend_radius_m)
    |   movel([0.427962, -1.438237, -2.523757, -0.750395, 1.570796, 1.998758],accel_mss,speed_ms,0,blend_radius_m)
    |   movel([0.428177, -1.437749, -2.524143, -0.750497, 1.570796, 1.998973],accel_mss,speed_ms,0,blend_radius_m)
    |   movel([0.428050, -1.436652, -2.525010, -0.750726, 1.570796, 1.998846],accel_mss,speed_ms,0,blend_radius_m)
    |   movel([0.427303, -1.435428, -2.525976, -0.750985, 1.570796, 1.998099],accel_mss,speed_ms,0,blend_radius_m)
    |   movel([0.424531, -1.432742, -2.528087, -0.751560, 1.570796, 1.995327],accel_mss,speed_ms,0,blend_radius_m)
    |   movel([0.421061, -1.429980, -2.530247, -0.752162, 1.570796, 1.991857],accel_mss,speed_ms,0,blend_radius_m)
    |   speed_ms = 0.003
    |   movel([0.421061, -1.423768, -2.527393, -0.761228, 1.570796, 1.991857],accel_mss,speed_ms,0,blend_radius_m)
    |   speed_ms = 0.05
    |   movel([0.421061, -1.399780, -2.515689, -0.796920, 1.570796, 1.991857],accel_mss,speed_ms,0,blend_radius_m)
    |   #M_RunCode9
    |   movel([0.554710, -1.326724, -2.566424, -0.819241, 1.570796, 2.125506],accel_mss,speed_ms,0,blend_radius_m)
    |   #M_RunCode3
    |   movel([0.554710, -1.352053, -2.579049, -0.781287, 1.570796, 2.125506],accel_mss,speed_ms,0,blend_radius_m)
    |   speed_ms = 0.003
    |   movel([0.554710, -1.358642, -2.582134, -0.771613, 1.570796, 2.125506],accel_mss,speed_ms,0,blend_radius_m)
    |   speed_ms = 0.02
    |   movel([0.554802, -1.357701, -2.582769, -0.771919, 1.570796, 2.125598],accel_mss,speed_ms,0,blend_radius_m)
    |   movel([0.555532, -1.356771, -2.583396, -0.772222, 1.570796, 2.126328],accel_mss,speed_ms,0,blend_radius_m)
    |   movel([0.555899, -1.356470, -2.583599, -0.772320, 1.570796, 2.126695],accel_mss,speed_ms,0,blend_radius_m)
    |   movel([0.558697, -1.354155, -2.585154, -0.773080, 1.570796, 2.129493],accel_mss,speed_ms,0,blend_radius_m)
    |   movel([0.561464, -1.351679, -2.586808, -0.773902, 1.570796, 2.132260],accel_mss,speed_ms,0,blend_radius_m)
    |   movel([0.563977, -1.349036, -2.588565, -0.774788, 1.570796, 2.134774],accel_mss,speed_ms,0,blend_radius_m)
    |   movel([0.566014, -1.346218, -2.590428, -0.775744, 1.570796, 2.136810],accel_mss,speed_ms,0,blend_radius_m)
    |   movel([0.567376, -1.343287, -2.592353, -0.776749, 1.570796, 2.138172],accel_mss,speed_ms,0,blend_radius_m)
    |   movel([0.568152, -1.340341, -2.594277, -0.777771, 1.570796, 2.138948],accel_mss,speed_ms,0,blend_radius_m)
    |   movel([0.568536, -1.337440, -2.596160, -0.778789, 1.570796, 2.139332],accel_mss,speed_ms,0,blend_radius_m)
    |   movel([0.568716, -1.334650, -2.597960, -0.779780, 1.570796, 2.139512],accel_mss,speed_ms,0,blend_radius_m)
    |   movel([0.568735, -1.334263, -2.598209, -0.779918, 1.570796, 2.139532],accel_mss,speed_ms,0,blend_radius_m)
    |   movel([0.569144, -1.333245, -2.598862, -0.780282, 1.570796, 2.139941],accel_mss,speed_ms,0,blend_radius_m)
    |   movel([0.570115, -1.332393, -2.599408, -0.780588, 1.570796, 2.140912],accel_mss,speed_ms,0,blend_radius_m)
    |   movel([0.571236, -1.332054, -2.599625, -0.780710, 1.570796, 2.142032],accel_mss,speed_ms,0,blend_radius_m)
    |   movel([0.572031, -1.332387, -2.599412, -0.780590, 1.570796, 2.142827],accel_mss,speed_ms,0,blend_radius_m)
    |   movel([0.572227, -1.332631, -2.599255, -0.780502, 1.570796, 2.143023],accel_mss,speed_ms,0,blend_radius_m)
    |   movel([0.573737, -1.334476, -2.598072, -0.779842, 1.570796, 2.144534],accel_mss,speed_ms,0,blend_radius_m)
    |   movel([0.575448, -1.336208, -2.596956, -0.779225, 1.570796, 2.146244],accel_mss,speed_ms,0,blend_radius_m)
    |   movel([0.577469, -1.337597, -2.596058, -0.778734, 1.570796, 2.148265],accel_mss,speed_ms,0,blend_radius_m)
    |   movel([0.579913, -1.338413, -2.595529, -0.778446, 1.570796, 2.150709],accel_mss,speed_ms,0,blend_radius_m)
    |   movel([0.582798, -1.338490, -2.595479, -0.778419, 1.570796, 2.153594],accel_mss,speed_ms,0,blend_radius_m)
    |   movel([0.585962, -1.337973, -2.595815, -0.778602, 1.570796, 2.156758],accel_mss,speed_ms,0,blend_radius_m)
    |   movel([0.589241, -1.337085, -2.596389, -0.778915, 1.570796, 2.160038],accel_mss,speed_ms,0,blend_radius_m)
    |   movel([0.592481, -1.336048, -2.597059, -0.779282, 1.570796, 2.163277],accel_mss,speed_ms,0,blend_radius_m)
    |   movel([0.592928, -1.335901, -2.597154, -0.779334, 1.570796, 2.163724],accel_mss,speed_ms,0,blend_radius_m)
    |   movel([0.593940, -1.335872, -2.597172, -0.779344, 1.570796, 2.164736],accel_mss,speed_ms,0,blend_radius_m)
    |   movel([0.594481, -1.336486, -2.596776, -0.779127, 1.570796, 2.165277],accel_mss,speed_ms,0,blend_radius_m)
    |   movel([0.594341, -1.337472, -2.596139, -0.778778, 1.570796, 2.165137],accel_mss,speed_ms,0,blend_radius_m)
    |   movel([0.593564, -1.338421, -2.595524, -0.778444, 1.570796, 2.164360],accel_mss,speed_ms,0,blend_radius_m)
    |   movel([0.593186, -1.338720, -2.595330, -0.778339, 1.570796, 2.163982],accel_mss,speed_ms,0,blend_radius_m)
    |   movel([0.590283, -1.341045, -2.593818, -0.777526, 1.570796, 2.161080],accel_mss,speed_ms,0,blend_radius_m)
    |   movel([0.587428, -1.343524, -2.592198, -0.776667, 1.570796, 2.158225],accel_mss,speed_ms,0,blend_radius_m)
    |   movel([0.584849, -1.346162, -2.590464, -0.775762, 1.570796, 2.155645],accel_mss,speed_ms,0,blend_radius_m)
    |   movel([0.582765, -1.348968, -2.588610, -0.774811, 1.570796, 2.153561],accel_mss,speed_ms,0,blend_radius_m)
    |   movel([0.581371, -1.351871, -2.586680, -0.773838, 1.570796, 2.152167],accel_mss,speed_ms,0,blend_radius_m)
    |   movel([0.580562, -1.354771, -2.584740, -0.772877, 1.570796, 2.151359],accel_mss,speed_ms,0,blend_radius_m)
    |   movel([0.580149, -1.357608, -2.582832, -0.771949, 1.570796, 2.150945],accel_mss,speed_ms,0,blend_radius_m)
    |   movel([0.579938, -1.360321, -2.580996, -0.771072, 1.570796, 2.150734],accel_mss,speed_ms,0,blend_radius_m)
    |   movel([0.579909, -1.360725, -2.580722, -0.770942, 1.570796, 2.150705],accel_mss,speed_ms,0,blend_radius_m)
    |   movel([0.579902, -1.360763, -2.580696, -0.770930, 1.570796, 2.150699],accel_mss,speed_ms,0,blend_radius_m)
    |   movel([0.579878, -1.360909, -2.580597, -0.770883, 1.570796, 2.150674],accel_mss,speed_ms,0,blend_radius_m)
    |   movel([0.579426, -1.361785, -2.580001, -0.770603, 1.570796, 2.150222],accel_mss,speed_ms,0,blend_radius_m)
    |   movel([0.578553, -1.362468, -2.579536, -0.770385, 1.570796, 2.149349],accel_mss,speed_ms,0,blend_radius_m)
    |   movel([0.577595, -1.362778, -2.579324, -0.770286, 1.570796, 2.148392],accel_mss,speed_ms,0,blend_radius_m)
    |   movel([0.576854, -1.362562, -2.579472, -0.770355, 1.570796, 2.147650],accel_mss,speed_ms,0,blend_radius_m)
    |   movel([0.576755, -1.362471, -2.579534, -0.770384, 1.570796, 2.147551],accel_mss,speed_ms,0,blend_radius_m)
    |   movel([0.576736, -1.362455, -2.579545, -0.770389, 1.570796, 2.147532],accel_mss,speed_ms,0,blend_radius_m)
    |   movel([0.576705, -1.362417, -2.579571, -0.770401, 1.570796, 2.147501],accel_mss,speed_ms,0,blend_radius_m)
    |   movel([0.576537, -1.362197, -2.579721, -0.770471, 1.570796, 2.147333],accel_mss,speed_ms,0,blend_radius_m)
    |   movel([0.575082, -1.360399, -2.580943, -0.771047, 1.570796, 2.145878],accel_mss,speed_ms,0,blend_radius_m)
    |   movel([0.573419, -1.358708, -2.582089, -0.771592, 1.570796, 2.144215],accel_mss,speed_ms,0,blend_radius_m)
    |   movel([0.571437, -1.357354, -2.583004, -0.772032, 1.570796, 2.142233],accel_mss,speed_ms,0,blend_radius_m)
    |   movel([0.569030, -1.356562, -2.583537, -0.772290, 1.570796, 2.139826],accel_mss,speed_ms,0,blend_radius_m)
    |   movel([0.566194, -1.356502, -2.583577, -0.772310, 1.570796, 2.136990],accel_mss,speed_ms,0,blend_radius_m)
    |   movel([0.563087, -1.357035, -2.583218, -0.772136, 1.570796, 2.133884],accel_mss,speed_ms,0,blend_radius_m)
    |   movel([0.559875, -1.357943, -2.582606, -0.771840, 1.570796, 2.130671],accel_mss,speed_ms,0,blend_radius_m)
    |   movel([0.556716, -1.359004, -2.581889, -0.771496, 1.570796, 2.127513],accel_mss,speed_ms,0,blend_radius_m)
    |   movel([0.556271, -1.359158, -2.581784, -0.771447, 1.570796, 2.127067],accel_mss,speed_ms,0,blend_radius_m)
    |   movel([0.555642, -1.359269, -2.581710, -0.771411, 1.570796, 2.126438],accel_mss,speed_ms,0,blend_radius_m)
    |   movel([0.555130, -1.359152, -2.581789, -0.771449, 1.570796, 2.125926],accel_mss,speed_ms,0,blend_radius_m)
    |   movel([0.554710, -1.358642, -2.582134, -0.771613, 1.570796, 2.125506],accel_mss,speed_ms,0,blend_radius_m)
    |   speed_ms = 0.003
    |   movel([0.554710, -1.352053, -2.579049, -0.781287, 1.570796, 2.125506],accel_mss,speed_ms,0,blend_radius_m)
    |   speed_ms = 0.05
    |   movel([0.554710, -1.326724, -2.566424, -0.819241, 1.570796, 2.125506],accel_mss,speed_ms,0,blend_radius_m)
    |   #M_RunCode9
    |   movel([0.347743, -1.354090, -2.548268, -0.810031, 1.570796, 1.918540],accel_mss,speed_ms,0,blend_radius_m)
    |   #M_RunCode3
    |   movel([0.347743, -1.378940, -2.560543, -0.772906, 1.570796, 1.918540],accel_mss,speed_ms,0,blend_radius_m)
    |   speed_ms = 0.003
    |   movel([0.347743, -1.385392, -2.563540, -0.763457, 1.570796, 1.918540],accel_mss,speed_ms,0,blend_radius_m)
    |   speed_ms = 0.02
    |   movel([0.347364, -1.386053, -2.563068, -0.763268, 1.570796, 1.918160],accel_mss,speed_ms,0,blend_radius_m)
    |   movel([0.347148, -1.386281, -2.562905, -0.763203, 1.570796, 1.917944],accel_mss,speed_ms,0,blend_radius_m)
    |   movel([0.343903, -1.389900, -2.560306, -0.762183, 1.570796, 1.914699],accel_mss,speed_ms,0,blend_radius_m)
    |   movel([0.342539, -1.391803, -2.558933, -0.761654, 1.570796, 1.913336],accel_mss,speed_ms,0,blend_radius_m)
    |   movel([0.341566, -1.393733, -2.557534, -0.761123, 1.570796, 1.912363],accel_mss,speed_ms,0,blend_radius_m)
    |   movel([0.341108, -1.395621, -2.556160, -0.760608, 1.570796, 1.911905],accel_mss,speed_ms,0,blend_radius_m)
    |   movel([0.341077, -1.397426, -2.554842, -0.760121, 1.570796, 1.911874],accel_mss,speed_ms,0,blend_radius_m)
    |   movel([0.341686, -1.400756, -2.552398, -0.759235, 1.570796, 1.912482],accel_mss,speed_ms,0,blend_radius_m)
    |   movel([0.341742, -1.400997, -2.552220, -0.759172, 1.570796, 1.912539],accel_mss,speed_ms,0,blend_radius_m)
    |   movel([0.341743, -1.401019, -2.552204, -0.759166, 1.570796, 1.912540],accel_mss,speed_ms,0,blend_radius_m)
    |   movel([0.341753, -1.401108, -2.552138, -0.759143, 1.570796, 1.912549],accel_mss,speed_ms,0,blend_radius_m)
    |   movel([0.341593, -1.401688, -2.551711, -0.758990, 1.570796, 1.912389],accel_mss,speed_ms,0,blend_radius_m)
    |   movel([0.341086, -1.402214, -2.551322, -0.758853, 1.570796, 1.911883],accel_mss,speed_ms,0,blend_radius_m)
    |   movel([0.340447, -1.402536, -2.551085, -0.758769, 1.570796, 1.911244],accel_mss,speed_ms,0,blend_radius_m)
    |   movel([0.339866, -1.402516, -2.551099, -0.758774, 1.570796, 1.910662],accel_mss,speed_ms,0,blend_radius_m)
    |   movel([0.339776, -1.402479, -2.551127, -0.758783, 1.570796, 1.910573],accel_mss,speed_ms,0,blend_radius_m)
    |   movel([0.339759, -1.402471, -2.551133, -0.758785, 1.570796, 1.910555],accel_mss,speed_ms,0,blend_radius_m)
    |   movel([0.339729, -1.402454, -2.551145, -0.758790, 1.570796, 1.910526],accel_mss,speed_ms,0,blend_radius_m)
    |   movel([0.339563, -1.402350, -2.551222, -0.758817, 1.570796, 1.910360],accel_mss,speed_ms,0,blend_radius_m)
    |   movel([0.336630, -1.400759, -2.552395, -0.759234, 1.570796, 1.907426],accel_mss,speed_ms,0,blend_radius_m)
    |   movel([0.334932, -1.400252, -2.552769, -0.759368, 1.570796, 1.905729],accel_mss,speed_ms,0,blend_radius_m)
    |   movel([0.333034, -1.400136, -2.552854, -0.759399, 1.570796, 1.903831],accel_mss,speed_ms,0,blend_radius_m)
    |   movel([0.330964, -1.400505, -2.552582, -0.759301, 1.570796, 1.901760],accel_mss,speed_ms,0,blend_radius_m)
    |   movel([0.328811, -1.401258, -2.552028, -0.759103, 1.570796, 1.899607],accel_mss,speed_ms,0,blend_radius_m)
    |   movel([0.324557, -1.403304, -2.550516, -0.758568, 1.570796, 1.895354],accel_mss,speed_ms,0,blend_radius_m)
    |   movel([0.324265, -1.403455, -2.550405, -0.758529, 1.570796, 1.895062],accel_mss,speed_ms,0,blend_radius_m)
    |   movel([0.323437, -1.403611, -2.550289, -0.758489, 1.570796, 1.894233],accel_mss,speed_ms,0,blend_radius_m)
    |   movel([0.323038, -1.403373, -2.550466, -0.758551, 1.570796, 1.893834],accel_mss,speed_ms,0,blend_radius_m)
    |   movel([0.322929, -1.402809, -2.550883, -0.758697, 1.570796, 1.893726],accel_mss,speed_ms,0,blend_radius_m)
    |   movel([0.323286, -1.402166, -2.551358, -0.758865, 1.570796, 1.894082],accel_mss,speed_ms,0,blend_radius_m)
    |   movel([0.323497, -1.401937, -2.551527, -0.758925, 1.570796, 1.894293],accel_mss,speed_ms,0,blend_radius_m)
    |   movel([0.326631, -1.398367, -2.554153, -0.759869, 1.570796, 1.897427],accel_mss,speed_ms,0,blend_radius_m)
    |   movel([0.327957, -1.396475, -2.555537, -0.760377, 1.570796, 1.898753],accel_mss,speed_ms,0,blend_radius_m)
    |   movel([0.328900, -1.394554, -2.556937, -0.760898, 1.570796, 1.899696],accel_mss,speed_ms,0,blend_radius_m)
    |   movel([0.329332, -1.392669, -2.558305, -0.761415, 1.570796, 1.900129],accel_mss,speed_ms,0,blend_radius_m)
    |   movel([0.329339, -1.390860, -2.559614, -0.761915, 1.570796, 1.900135],accel_mss,speed_ms,0,blend_radius_m)
    |   movel([0.328671, -1.387512, -2.562023, -0.762854, 1.570796, 1.899468],accel_mss,speed_ms,0,blend_radius_m)
    |   movel([0.328612, -1.387288, -2.562184, -0.762917, 1.570796, 1.899409],accel_mss,speed_ms,0,blend_radius_m)
    |   movel([0.328714, -1.386646, -2.562643, -0.763099, 1.570796, 1.899510],accel_mss,speed_ms,0,blend_radius_m)
    |   movel([0.329251, -1.386021, -2.563091, -0.763277, 1.570796, 1.900048],accel_mss,speed_ms,0,blend_radius_m)
    |   movel([0.329994, -1.385666, -2.563344, -0.763378, 1.570796, 1.900791],accel_mss,speed_ms,0,blend_radius_m)
    |   movel([0.330631, -1.385743, -2.563289, -0.763356, 1.570796, 1.901427],accel_mss,speed_ms,0,blend_radius_m)
    |   movel([0.330819, -1.385856, -2.563209, -0.763324, 1.570796, 1.901615],accel_mss,speed_ms,0,blend_radius_m)
    |   movel([0.333822, -1.387439, -2.562075, -0.762874, 1.570796, 1.904618],accel_mss,speed_ms,0,blend_radius_m)
    |   movel([0.335550, -1.387944, -2.561713, -0.762732, 1.570796, 1.906346],accel_mss,speed_ms,0,blend_radius_m)
    |   movel([0.337473, -1.388057, -2.561632, -0.762700, 1.570796, 1.908270],accel_mss,speed_ms,0,blend_radius_m)
    |   movel([0.339574, -1.387682, -2.561901, -0.762806, 1.570796, 1.910371],accel_mss,speed_ms,0,blend_radius_m)
    |   movel([0.341766, -1.386920, -2.562447, -0.763022, 1.570796, 1.912562],accel_mss,speed_ms,0,blend_radius_m)
    |   movel([0.346116, -1.384852, -2.563926, -0.763611, 1.570796, 1.916913],accel_mss,speed_ms,0,blend_radius_m)
    |   movel([0.346413, -1.384702, -2.564033, -0.763654, 1.570796, 1.917209],accel_mss,speed_ms,0,blend_radius_m)
    |   movel([0.347140, -1.384535, -2.564151, -0.763702, 1.570796, 1.917936],accel_mss,speed_ms,0,blend_radius_m)
    |   movel([0.347651, -1.384806, -2.563958, -0.763624, 1.570796, 1.918447],accel_mss,speed_ms,0,blend_radius_m)
    |   movel([0.347743, -1.385392, -2.563540, -0.763457, 1.570796, 1.918540],accel_mss,speed_ms,0,blend_radius_m)
    |   speed_ms = 0.003
    |   movel([0.347743, -1.378940, -2.560543, -0.772906, 1.570796, 1.918540],accel_mss,speed_ms,0,blend_radius_m)
    |   speed_ms = 0.05
    |   movel([0.347743, -1.354090, -2.548268, -0.810031, 1.570796, 1.918540],accel_mss,speed_ms,0,blend_radius_m)
    |   #M_RunCode9
    |   movel([0.369740, -1.091711, -2.685705, -0.934973, 1.570796, 1.940536],accel_mss,speed_ms,0,blend_radius_m)
    |   movel([0.369740, -1.032662, -2.644702, -1.035025, 1.570796, 1.940536],accel_mss,speed_ms,0,blend_radius_m)
    |   #M_RunCode2
    |   # End of main program
    | end
    | 
    | Machining1()
